// TIA Portal V19 export
FUNCTION "FC_AEND_WT" : Void   // FC45, STL
TITLE = WT-Daten neu/geändert
{ S7_Optimized_Access := 'FALSE' }
AUTHOR : MS
// Laden von WT-Daten aus Übergabepuffer
// stored: AutoNumber false
   VAR_TEMP
      WT_lang : DWord;
      WT_Nr_lang : DWord;
      WT_DB : Int;
      Quell_DB : Int;
      last_WT_DB : Int;
      Beginn_Daten : Int;
      Ende_daten : Int;
      Stand_Nr : USInt;
      Pos_Nr : USInt;
      WT_Nr : Byte;
      WT_kurz : Byte;
      inf_1 : Byte;
      WTnew : Bool;   // Warenträger neu
      "Return" : Bool;
      Stand_ok : Bool;
      WT_nok : Bool;
      neuAufgabe : Bool;
      Del_All : Bool;
   END_VAR
BEGIN

NETWORK
TITLE = Test gibt es neue Daten
// -gibt es neue Daten
// -wo stehen diese
// -handelt es sich um Aktualisierungsdaten
//-------------------------------
//Neue Daten?
//-------------------------------
      A     "DB_Techno".DATEN_gueltig;
      L     S5T#20S;
      SD    "T_Aend_WT";

      A     "DB_Techno".DATEN_gueltig;
      A     "T_Aend_WT";
      R     "DB_Techno".DATEN_gueltig;
//-------------------------------
//keine neuen Daten
//-------------------------------
      AN    "DB_Techno".DATEN_gueltig;
      BEC;
      SET;
      R     #Stand_ok;
      R     #Del_All;

//----------------------------------
//Handelt es sich um eine Neuaufgabe
//----------------------------------
      L     "DB_Techno".STAND_NR;
      T     #Stand_Nr;
      L     0;
      <>I;
      =     #WTnew;
      =     #neuAufgabe;
      JC    New;
      JU    Old;


NETWORK
TITLE = Neuer WT
//------------------------
//Stand-Nr prüfen
//------------------------
New:  L     "DB_BE_Stand".Anzahl;
      L     #Stand_Nr;
      <I;
      JC    ende;

      OPN   "DB_BE_Stand";
      A     "DB_BE_Stand".Stand[#Stand_Nr].Del_All;
      =     #Del_All;
      L     0;
      L     "DB_BE_Stand".Stand[#Stand_Nr].Pos_Nr;
      ==I;
      JC    ende;
      S     #Stand_ok;
//------------------------
//Pos auf WT testen
//------------------------
      T     #Pos_Nr;
      L     0;
      L     "DB_POS".POS[#Pos_Nr].WT_DB;
      ==I;
      JC    WTck;
      T     #WT_Nr;
      L     100;
      +I;
      T     #WT_DB;
      JU    load;
//------------------------
//Neuen WT suchen
//------------------------
WTck: AN    #Del_All;  //keinen neuen WT suchen
      JC    ende;
      L     "DB_ANLAGE".config.ANZ_WT;
      L     100;
      +I;
      T     #last_WT_DB;
      L     101;
      T     #WT_DB;
ret:  OPN   DB [#WT_DB];
      L     %DBB15;
      L     0;
      ==I;
      JC    fnd;
      L     #WT_DB;
      L     1;
      +I;
      T     #WT_DB;
      L     #last_WT_DB;
      >I;
      JC    ende;
      JU    ret;
fnd:  L     #WT_DB;
      L     100;
      -I;
      T     #WT_Nr;
      JU    load;


NETWORK
TITLE = Alter WT
// Aktualisieren
//-------------------------------
//prüfen ob WT_Nr gültig
//-------------------------------
Old:  L     "DB_Techno".WT_NR_kurz;
      T     #WT_Nr;
      L     "DB_ANLAGE".config.ANZ_WT;
      >I;
      JC    ende;
      L     0;
      L     #WT_Nr;
      >=I;
      JC    ende;
      L     100;
      +I;
      T     #WT_DB;
//-------------------------------
//passen die WT-Daten zueinander
//-------------------------------
      L     "DB_Techno".WT_NR_lng;
      OPN   DB [#WT_DB];
      L     %DBD6;  // WT-Nr lang
      <>D;
      JC    ende;
      L     %DBB15;  //"DB_WTx".POS
      T     #Pos_Nr;

load: NOP   0;

NETWORK
TITLE = Daten laden
//------------------------
//allgemeine Daten laden
//------------------------
ldok: L     "DB_Techno".Beginn_Daten;
      T     #Beginn_Daten;
      L     "DB_Techno".Ende_Daten;
      T     #Ende_daten;

      CALL  "FC_DB_COPY"
      ( CLR_ALT_DB := FALSE,
        ALT_DB     := 45,
        NEU_DB     := #WT_DB,
        COPY_START := #Beginn_Daten,
        COPY_ENDE  := #Ende_daten,
        ZIEL_START := 78,  // HCA: Namen mit kopieren
        CLR_START  := 0,
        CLR_ENDE   := 0,
        START      := "DB_Techno".DATEN_gueltig
      );

      L     "DB_Techno".Prioritaet;
      L     0;
      <>I;
      OPN   DB [#WT_DB];
      =     %DBX18.0;  //PRIORITÄT

      OPN   DB [#WT_DB];
      A     %DBX18.1;  //"DB_WT1".in_Anlage
      R     #neuAufgabe;  //WT wurde bereits neu aufgegeben

      A     %DBX22.3;  //"DB_WT1".WT_nok
      AN    #Stand_ok;
      =     #WT_nok;  //nok merken

      L     "DB_Techno".ParaByte;  //Parameterinfo laden
      OPN   DB [#WT_DB];
      T     %DBB22;
      L     "DB_Techno".WT_NR_lng;
      OPN   DB [#WT_DB];
      T     %DBD6;  //WT_Nr_lang
      T     #WT_Nr_lang;
      L     "DB_Techno".Speed_Up;
      OPN   DB [#WT_DB];
      T     %DBW64;  //"DB_WT1".Speed_Up
      L     "DB_Techno".Speed_Dn;
      OPN   DB [#WT_DB];
      T     %DBW66;  //"DB_WT1".Speed_Dn
      L     "DB_Techno".Speed_Fahrt;
      OPN   DB [#WT_DB];
      T     %DBW68;  //"DB_WT1".Speed_Fahrt
      L     "DB_Techno".KorrPend;  //Korrektur Pendeln laden
      OPN   DB [#WT_DB];
      T     %DBD38;
      L     "DB_Techno".KorrATZ;  //Korrektur Tropfen laden
      OPN   DB [#WT_DB];
      T     %DBD42;
      L     "DB_Techno".WT_Kennung;
      OPN   DB [#WT_DB];
      T     %DBB63;
      L     "DB_Techno".WT_Typ;
      OPN   DB [#WT_DB];
      T     %DBB35;

      OPN   DB [#WT_DB];
      A     #WT_nok;  //nok zurückladen
      =     %DBX22.3;  //"DB_WT1".WT_nok

      CALL  "FC_TechScan"
      ( WT_DB_Nr := #WT_DB
      );

      AN    #WTnew;
      JC    OEvt;
//------------------------
//Daten bei neuem WT
//------------------------

      L     "DB_Techno".Oberflaeche;
      OPN   DB [#WT_DB];
      T     %DBD10;
      L     0;
      T     %DBW46;  //Parameterpointer
      T     %DBW48;  //Befehlspointer
      T     %DBB20;  //Behandlungsbits
      T     %DBD30;  //"DB_WT1".Fertigzeitpunkt

      L     "DB_Techno".Korb_Nr;
      OPN   DB [#WT_DB];
      T     %DBB14;  //"DB_WTx".Korb_Nr

      CALL  "FC_Korbumlaeufe"
      ( Nr := "DB_Techno".Korb_Nr
      );

      L     "DB_Techno".Technologie;
      OPN   DB [#WT_DB];
      T     %DBW16;  //Technologienummer
      OPN   DB [#WT_DB];
      L     #Pos_Nr;
      T     %DBB15;  //WT Ist-Pos
      T     %DBB19;  //WT Auto-Pos

      L     "DB_Panel_OVERVIEW".Systime;
      OPN   DB [#WT_DB];
      T     %DBD74;  //"DB_WT1".Aufgabezeit

      SET;
      R     %DBX20.0;  //Trommel
      S     %DBX18.1;  //in Anlage
      R     %DBX18.2;  //in Entmetallisierung
      R     %DBX18.3;  //aus Anlage
      R     %DBX18.4;  //aus Entmetallisierung
      R     %DBX18.5;  //Speicherprogramm


NETWORK
TITLE = 
// WT in Position laden
      CALL  "FC_WT_to_Pos"
      ( Pos_Nr     := #Pos_Nr,
        WT_Nr      := #WT_Nr,
        BA_Auto    := TRUE,
        send_DBEvt := FALSE,
        SimLoad    := FALSE,
        Copy_ok    := #"Return"
      );

// Langware in beide Positionen laden

      L     "DB_Techno".WT_Typ;
      L     b#16#12;  //Lang schmal
      <>I;
      JC    ende;
      L     #Pos_Nr;
      INC   1;
      T     #Pos_Nr;

      CALL  "FC_WT_to_Pos"
      ( Pos_Nr     := #Pos_Nr,
        WT_Nr      := #WT_Nr,
        BA_Auto    := TRUE,
        send_DBEvt := FALSE,
        SimLoad    := FALSE,
        Copy_ok    := #"Return"
      );

      JU    ende;

OEvt: NOP   0;

      CALL  "FC_WT_from_Pos"
      ( Pos_Nr     := #Pos_Nr,
        send_DBEvt := FALSE,
        load_ok    := #"Return",
        WT_Nr      := #WT_kurz,
        WT_Nr_lang := #WT_lang
      );

      AN    #"Return";
      JC    ende;

      CALL  "FC_WT_to_Pos"
      ( Pos_Nr     := #Pos_Nr,
        WT_Nr      := #WT_kurz,
        BA_Auto    := FALSE,
        send_DBEvt := FALSE,
        SimLoad    := FALSE,
        Copy_ok    := #"Return"
      );

ende: BE;

END_FUNCTION
